Universal Robots PolyScope program: 2_hover_to_gls_pick.urp

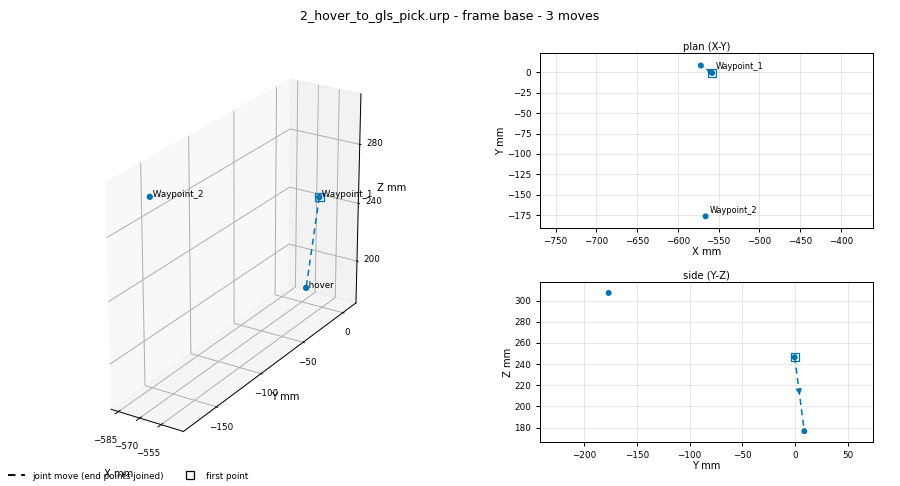
[picture p0: tool path of 2_hover_to_gls_pick.urp in frame base, 3 of 4 moves have a stored position in this frame; points joined in program order, loops and branches not executed]
Program 2_hover_to_gls_pick (installation=default directory=/programs/washer_rahman createdIn=5.9.5.1031259 lastSavedIn=5.9.5.1031259 robotSerialNumber=20215500597)
Calibrated DH parameters: a=[0.000193, -0.066673, -0.391568, -0.000012, 0.00005, 0]; d=[0.162643, -472.05677, 465.132521, 7.058239, 0.099746, 0.099582]; alpha=[1.571116, 0.00089, 0.003862, 1.569269, -1.569248, 0]; deltaTheta=[0, -1.413394, 7.628392, 0.068187, 0, -0.000001]
Robot Program (runOnlyOnce=true)
  SuppressedNode
    var_1 := 3
  SuppressedNode
    Script: glass_hover=p[-.603,-0.23+var_1*0.150 ,0.277,2.067,2.652,-2.043]
  Script: glass_hover=p[-.603,-0.23+GP_int_in[0]*0.150 ,0.277,2.067,2.652,-2.043]
  MoveJ speed 60 deg/s, acceleration 80 deg/s^2 (useActiveTCP=true) feature=Base
    Waypoint Waypoint_1: TCP in base x=-557.948 y=-0.617 z=246.473 mm, rx=-1.2337 ry=-1.2229 rz=1.2356 rad; joints [-31.234, -63.252, 147.704, -263.239, -57.852, 1.051] deg; TCP offset x=0 y=0 z=191.5 mm, rx=0 ry=0 rz=0 rad
  MoveJ speed 60 deg/s, acceleration 80 deg/s^2 (useActiveTCP=true) feature=Base
    Waypoint hover: TCP in base x=-571.891 y=8.47 z=176.529 mm, rx=-1.3535 ry=-1.4262 rz=1.0959 rad; joints [-31.225, -63.222, 147.699, -247.797, -58.006, -9.864] deg
  MoveL speed 250 mm/s, acceleration 1200 mm/s^2 (useActiveTCP=true) feature=Base
    MoveDirectionNode (selectedDirection=ZPlus)
      Until DISTANCE (allowActions=false deceleration=3 distanceNodeType=STOP) Distance=0.1; motionParameters(blendRadius=0)
    SuppressedNode
      MoveDirectionNode (selectedDirection=XMinus)
        Until DISTANCE (allowActions=false deceleration=3 distanceNodeType=STOP) Distance=0.08; motionParameters(blendRadius=0)
  MoveJ speed 60 deg/s, acceleration 80 deg/s^2 (useActiveTCP=true) feature=Base
    Waypoint Waypoint (Variable): variable=glass_hover
  MoveL speed 250 mm/s, acceleration 1200 mm/s^2 (useActiveTCP=true) feature=Base
    MoveDirectionNode (selectedDirection=ZMinus)
      Until DISTANCE (allowActions=false deceleration=3 distanceNodeType=STOP) Distance=0.18; motionParameters(blendRadius=0)
  URCap Gripper (Robotiq_Grippers, Robotiq Inc.) dataModel(position=31.372549019607842, force=0.0, speed=0.0, positionInDouble=31.372549019607842, forceInDouble=0.0, speedInDouble=0.0, slaveIds=[9], blocking=true)
  MoveL speed 250 mm/s, acceleration 1200 mm/s^2 (useActiveTCP=true) feature=Base
    MoveDirectionNode (selectedDirection=ZPlus)
      Until DISTANCE (allowActions=false deceleration=3 distanceNodeType=STOP) Distance=0.2; motionParameters(blendRadius=0)
  MoveJ speed 60 deg/s, acceleration 80 deg/s^2 (useActiveTCP=true) feature=Base
    Waypoint Waypoint_2: TCP in base x=-566.058 y=-176.538 z=307.302 mm, rx=-1.2228 ry=-1.3732 rz=1.1429 rad; joints [5.319, -79.632, 138.521, -231.601, -92.317, -3.014] deg
